TYPE ST_WierszListyRecepturDlaHMI :
STRUCT
	wsTekst			: WSTRING;
	iNumer			: INT;
	refReceptura	: reference to ST_Receptura;
END_STRUCT
END_TYPE

(* stored: Version 1.1.0.1
   DUT ST_WierszListyRecepturDlaHMI: Id {25f5150b-f32b-0a24-1a7a-4eedc0019634} *)
